SYSTEM Test Reader
  (* Version 1.0, 2005-06-27, Goran Cengic, Chalmers *)
  DEVICE Test Device : DeviceType_not_used
    RESOURCE TestResource : ResourceType_not_used
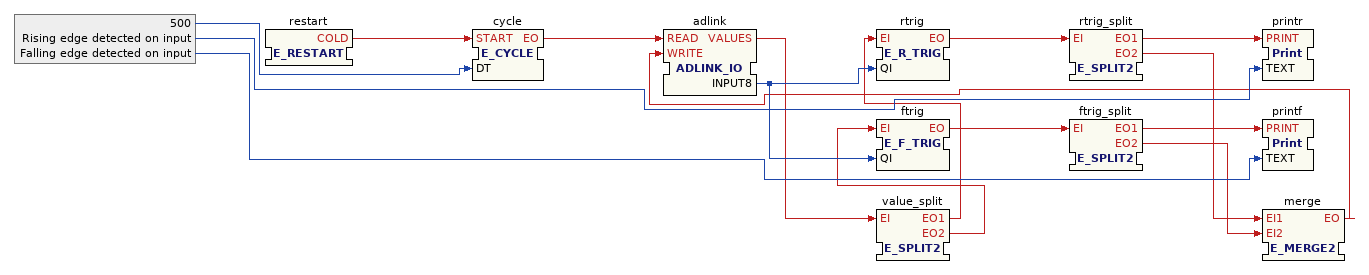
      FBS
        restart : E_RESTART;
        cycle : E_CYCLE;
        adlink : ADLINK_IO;
        rtrig : E_R_TRIG;
        ftrig : E_F_TRIG;
        value_split : E_SPLIT2;
        rtrig_split : E_SPLIT2;
        ftrig_split : E_SPLIT2;
        printr : Print;
        printf : Print;
        merge : E_MERGE2;
      END_FBS
      EVENT_CONNECTIONS
        restart.COLD TO cycle.START;
        cycle.EO TO adlink.READ;
        adlink.VALUES TO value_split.EI;
        value_split.EO1 TO rtrig.EI;
        value_split.EO2 TO ftrig.EI;
        rtrig.EO TO rtrig_split.EI;
        ftrig.EO TO ftrig_split.EI;
        rtrig_split.EO1 TO printr.PRINT;
        rtrig_split.EO2 TO merge.EI1;
        ftrig_split.EO1 TO printf.PRINT;
        ftrig_split.EO2 TO merge.EI2;
        merge.EO TO adlink.WRITE;
      END_CONNECTIONS
      DATA_CONNECTIONS
        500 TO cycle.DT;
        adlink.INPUT8 TO rtrig.QI;
        adlink.INPUT8 TO ftrig.QI;
        Rising edge detected on input TO printr.TEXT;
        Falling edge detected on input TO printf.TEXT;
      END_CONNECTIONS
    END_RESOURCE
  END_DEVICE
END_SYSTEM
(* other elements stored in the file *)
(* Connection Source="true" Destination="adlink.OUTPUT16" / *)
(* Connection Source="adlink.INPUT4" Destination="adlink.OUTPUT4" / *)
(* Connection Source="adlink.INPUT2" Destination="adlink.OUTPUT15" / *)
